{attribute 'qualified_only'}
{attribute 'global_init_slot' := '40550'}
VAR_GLOBAL
	arrElementyWykonawcze 					: ARRAY [1..GVL_LogowanieBledow_Stale.MAX_ILOSC_ELEMENTOW] OF 
																ITF_LogowanieBledow_ElementWykonawczy := [
																	GVL_Podzespoly.fbKrajalnica.fbLBKomunikacja];

	fbLoger 								: FB_LogowanieBledow (	tablica := arrElementyWykonawcze,
																	iIloscDodanychElementow := 1);
	bWyswietlAlarmy							: BOOL;																
	
END_VAR
VAR_GLOBAL //PERSISTENT
	arrTablicaZdarzenZapamietancyh			: ARRAY [1..GVL_LogowanieBledow_Stale.MAX_ILOSC_ZDARZEN_ZAPAMIETANYCH] OF DUT_LogowanieBledow_Zapamietanych;																
	
	iIloscZdarzenZapamietanych				: INT;	//ilosc zdarzen ktore wystapiły
END_VAR

(* stored: Version 1.1.0.1, ProductVersion 3.1.4024.11
   GVL GVL_LogowanieBledow: Id {031458d1-4327-4414-a5e1-6329ee0946ec} *)
